(* LS Electric XG5000 project: 232통신_테스트 *)
(* PLC NewPLC *)
(* module base 0 slot 0: FEnet:XGL-EFMT(B) (Fast Ethernet 통신 모듈, 전기 Master) *)
(* module base 0 slot 1: Cnet:XGL-CH2A/B (Cnet 통신 모듈(RS-232C, RS-422/485)) *)
(* module base 0 slot 2: 입력 모듈:XGI-D22A/B (DC 24V 입력, 16점 (전류소스 싱크공용/ 전류소스 입력)) *)
(* module base 0 slot 3: 출력 모듈:XGQ-RY2A/B (릴레이 출력, 16점 (2A용, Varistor 없음/Varistor 부착)) *)

PROGRAM 메인 (* task: 스캔 프로그램 *)
VAR
    timer : TON;
    WATER_TIMER : TON;
    남은금액_1 : UINT;
    남은금액_2 : UINT;
    반환_타이머 : BOOL;
    사이다_TIMER : TON;
    식혜_TIMER : TON;
    알로에_TIMER : TON;
    자판기_거스름돈갯수_100원 AT %MW123 : UINT; (* 자판기_거스름돈갯수_100원 *)
    자판기_거스름돈갯수_500원 AT %MW122 : UINT; (* 자판기_거스름돈갯수_500원 *)
    자판기_거스름돈갯수_50원 AT %MW124 : UINT; (* 자판기_거스름돈갯수_50원 *)
    자판기_금액투입_1000원 AT %MW100.0 : BOOL; (* 자판기_금액투입_1000원 *)
    자판기_금액투입_100원 AT %MW100.2 : BOOL; (* 자판기_금액투입_100원 *)
    자판기_금액투입_500원 AT %MW100.1 : BOOL; (* 자판기_금액투입_500원 *)
    자판기_금액투입_50원 AT %MW100.3 : BOOL; (* 자판기_금액투입_50원 *)
    자판기_남은금액 AT %MW121 : UINT; (* 자판기_남은금액 *)
    자판기_물구매_700원 AT %MW100.5 : BOOL; (* 자판기_물구매_700원 *)
    자판기_반환버튼 AT %MW100.4 : BOOL; (* 자판기_반환버튼 *)
    자판기_사이다구매_1000원 AT %MW100.6 : BOOL; (* 자판기_사이다구매_1000원 *)
    자판기_식혜구매_1200원 AT %MW100.8 : BOOL; (* 자판기_식혜구매_1200원 *)
    자판기_알로에구매_1300원 AT %MW100.9 : BOOL; (* 자판기_알로에구매_1300원 *)
    자판기_음료출몰_물 AT %MW110.4 : BOOL; (* 자판기_음료출몰_물 *)
    자판기_음료출몰_사이다 AT %MW110.5 : BOOL; (* 자판기_음료출몰_사이다 *)
    자판기_음료출몰_식혜 AT %MW110.7 : BOOL; (* 자판기_음료출몰_식혜 *)
    자판기_음료출몰_알로에 AT %MW110.8 : BOOL; (* 자판기_음료출몰_알로에 *)
    자판기_음료출몰_콜라 AT %MW110.6 : BOOL; (* 자판기_음료출몰_콜라 *)
    자판기_콜라구매_1000원 AT %MW100.7 : BOOL; (* 자판기_콜라구매_1000원 *)
    자판기_투입금액 AT %MW120 : UINT; (* 자판기_투입금액 *)
    자판기램프_물 AT %MW110.0 : BOOL; (* 자판기램프_물 *)
    자판기램프_사이다_콜라 AT %MW110.1 : BOOL; (* 자판기램프_사이다_콜라 *)
    자판기램프_식혜 AT %MW110.2 : BOOL; (* 자판기램프_식혜 *)
    자판기램프_알로에 AT %MW110.3 : BOOL; (* 자판기램프_알로에 *)
    콜라_TIMER : TON;
END_VAR
VAR
    _e1 : R_TRIG;
    _e2 : R_TRIG;
    _e3 : R_TRIG;
    _e4 : R_TRIG;
    _e5 : R_TRIG;
    _e6 : R_TRIG;
    _t7 : BOOL;
    _e8 : R_TRIG;
    _t9 : BOOL;
    _t10 : BOOL;
    _e11 : R_TRIG;
    _t12 : BOOL;
    _e13 : R_TRIG;
    _e14 : F_TRIG;
    _e15 : R_TRIG;
    _t16 : BOOL;
    _e17 : R_TRIG;
    _t18 : BOOL;
    _e19 : R_TRIG;
    _t20 : BOOL;
    _e21 : R_TRIG;
    _t22 : BOOL;
    _e23 : R_TRIG;
    _t24 : BOOL;
END_VAR

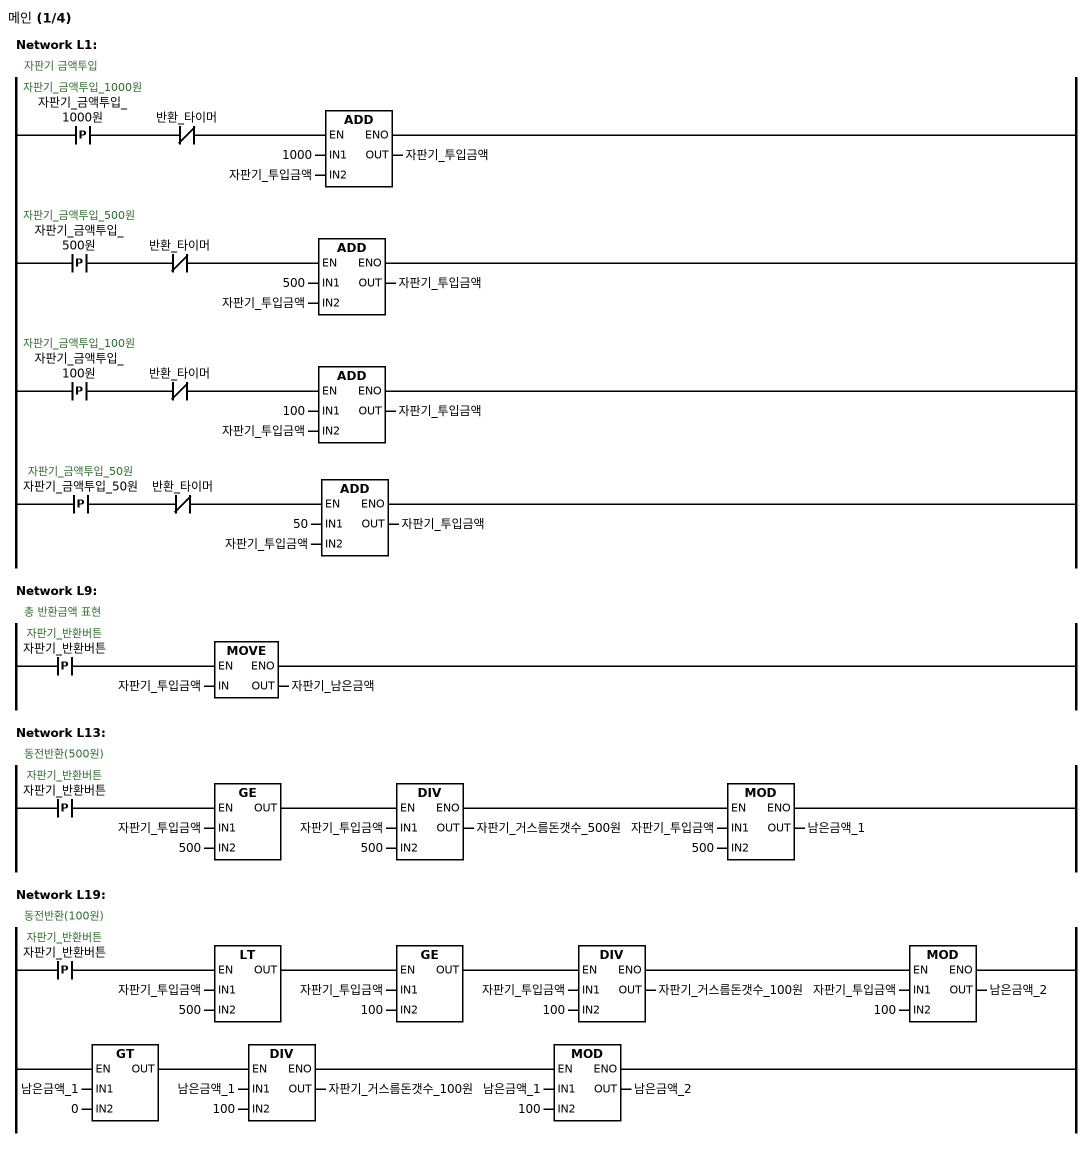
(* 자판기 금액투입 *)
(* Rung L1 *)
_e1(CLK := 자판기_금액투입_1000원);
IF _e1.Q AND NOT 반환_타이머 THEN 자판기_투입금액 := 1000 + 자판기_투입금액; END_IF;
_e2(CLK := 자판기_금액투입_500원);
IF _e2.Q AND NOT 반환_타이머 THEN 자판기_투입금액 := 500 + 자판기_투입금액; END_IF;
_e3(CLK := 자판기_금액투입_100원);
IF _e3.Q AND NOT 반환_타이머 THEN 자판기_투입금액 := 100 + 자판기_투입금액; END_IF;
_e4(CLK := 자판기_금액투입_50원);
IF _e4.Q AND NOT 반환_타이머 THEN 자판기_투입금액 := 50 + 자판기_투입금액; END_IF;
(* 총 반환금액 표현 *)
(* Rung L9 *)
_e5(CLK := 자판기_반환버튼);
IF _e5.Q THEN 자판기_남은금액 := 자판기_투입금액; END_IF;
(* 동전반환(500원) *)
(* Rung L13 *)
_e6(CLK := 자판기_반환버튼);
IF _e6.Q THEN _t7 := 자판기_투입금액 >= 500; END_IF;
IF _t7 THEN
    자판기_거스름돈갯수_500원 := 자판기_투입금액 / 500;
    남은금액_1 := 자판기_투입금액 MOD 500;
END_IF;
(* 동전반환(100원) *)
(* Rung L19 *)
_e8(CLK := 자판기_반환버튼);
IF _e8.Q THEN _t9 := 자판기_투입금액 < 500; END_IF;
IF _t9 THEN _t10 := 자판기_투입금액 >= 100; END_IF;
IF _t10 THEN
    자판기_거스름돈갯수_100원 := 자판기_투입금액 / 100;
    남은금액_2 := 자판기_투입금액 MOD 100;
END_IF;
IF 남은금액_1 > 0 THEN
    자판기_거스름돈갯수_100원 := 남은금액_1 / 100;
    남은금액_2 := 남은금액_1 MOD 100;
END_IF;

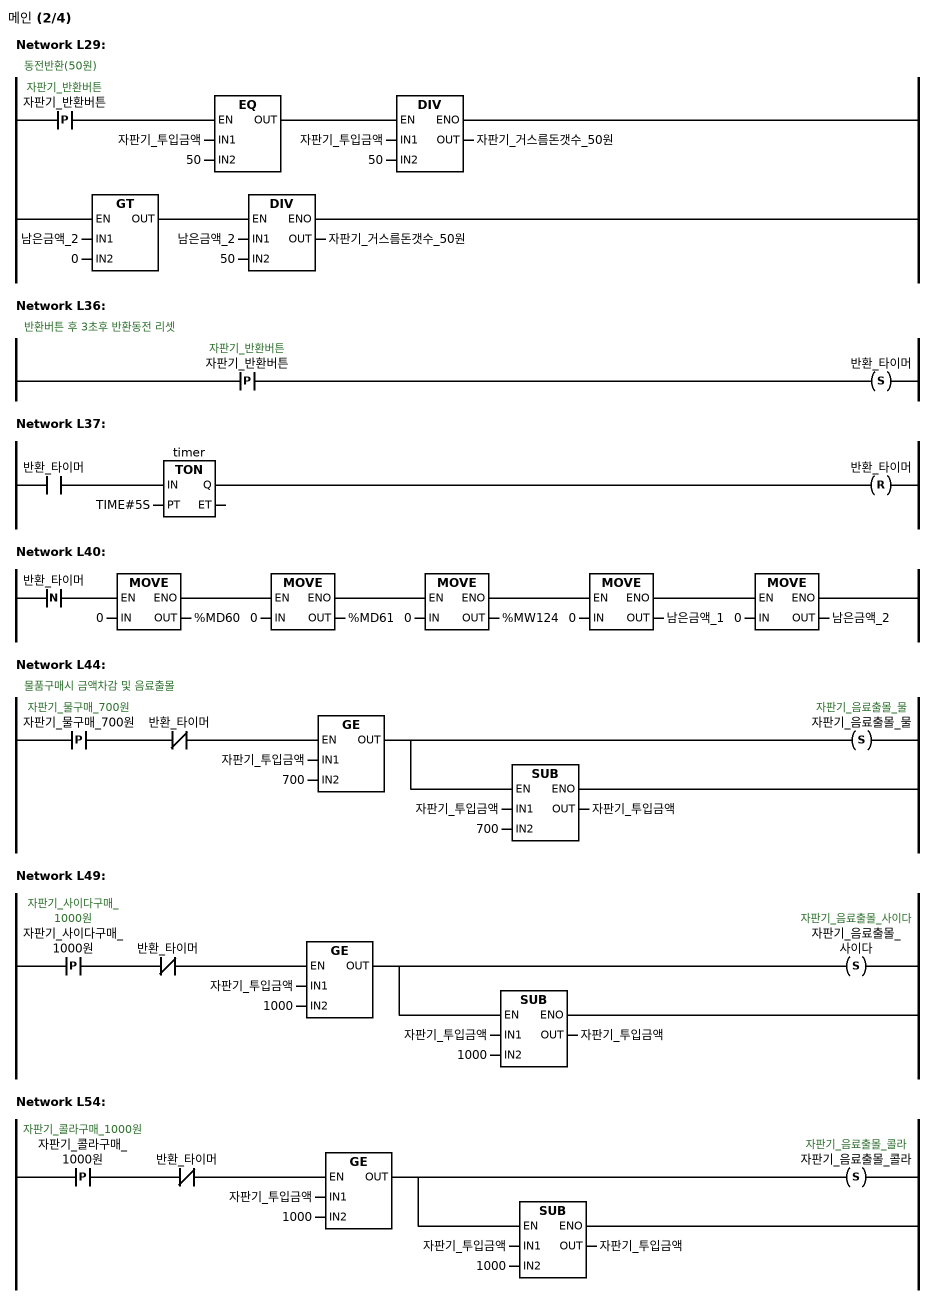
(* 동전반환(50원) *)
(* Rung L29 *)
_e11(CLK := 자판기_반환버튼);
IF _e11.Q THEN _t12 := 자판기_투입금액 = 50; END_IF;
IF _t12 THEN 자판기_거스름돈갯수_50원 := 자판기_투입금액 / 50; END_IF;
IF 남은금액_2 > 0 THEN 자판기_거스름돈갯수_50원 := 남은금액_2 / 50; END_IF;
(* 반환버튼 후 3초후 반환동전 리셋 *)
(* Rung L36 *)
_e13(CLK := 자판기_반환버튼);
IF _e13.Q THEN 반환_타이머 := TRUE; END_IF;
(* Rung L37 *)
timer(IN := 반환_타이머, PT := TIME#5S);
IF timer.Q THEN 반환_타이머 := FALSE; END_IF;
(* Rung L40 *)
_e14(CLK := 반환_타이머);
IF _e14.Q THEN
    %MD60 := 0;
    %MD61 := 0;
    %MW124 := 0;
    남은금액_1 := 0;
    남은금액_2 := 0;
END_IF;
(* 물품구매시 금액차감 및 음료출몰 *)
(* Rung L44 *)
_e15(CLK := 자판기_물구매_700원);
IF _e15.Q AND NOT 반환_타이머 THEN _t16 := 자판기_투입금액 >= 700; END_IF;
IF _t16 THEN
    자판기_음료출몰_물 := TRUE;
    자판기_투입금액 := 자판기_투입금액 - 700;
END_IF;
(* Rung L49 *)
_e17(CLK := 자판기_사이다구매_1000원);
IF _e17.Q AND NOT 반환_타이머 THEN _t18 := 자판기_투입금액 >= 1000; END_IF;
IF _t18 THEN
    자판기_음료출몰_사이다 := TRUE;
    자판기_투입금액 := 자판기_투입금액 - 1000;
END_IF;
(* Rung L54 *)
_e19(CLK := 자판기_콜라구매_1000원);
IF _e19.Q AND NOT 반환_타이머 THEN _t20 := 자판기_투입금액 >= 1000; END_IF;
IF _t20 THEN
    자판기_음료출몰_콜라 := TRUE;
    자판기_투입금액 := 자판기_투입금액 - 1000;
END_IF;

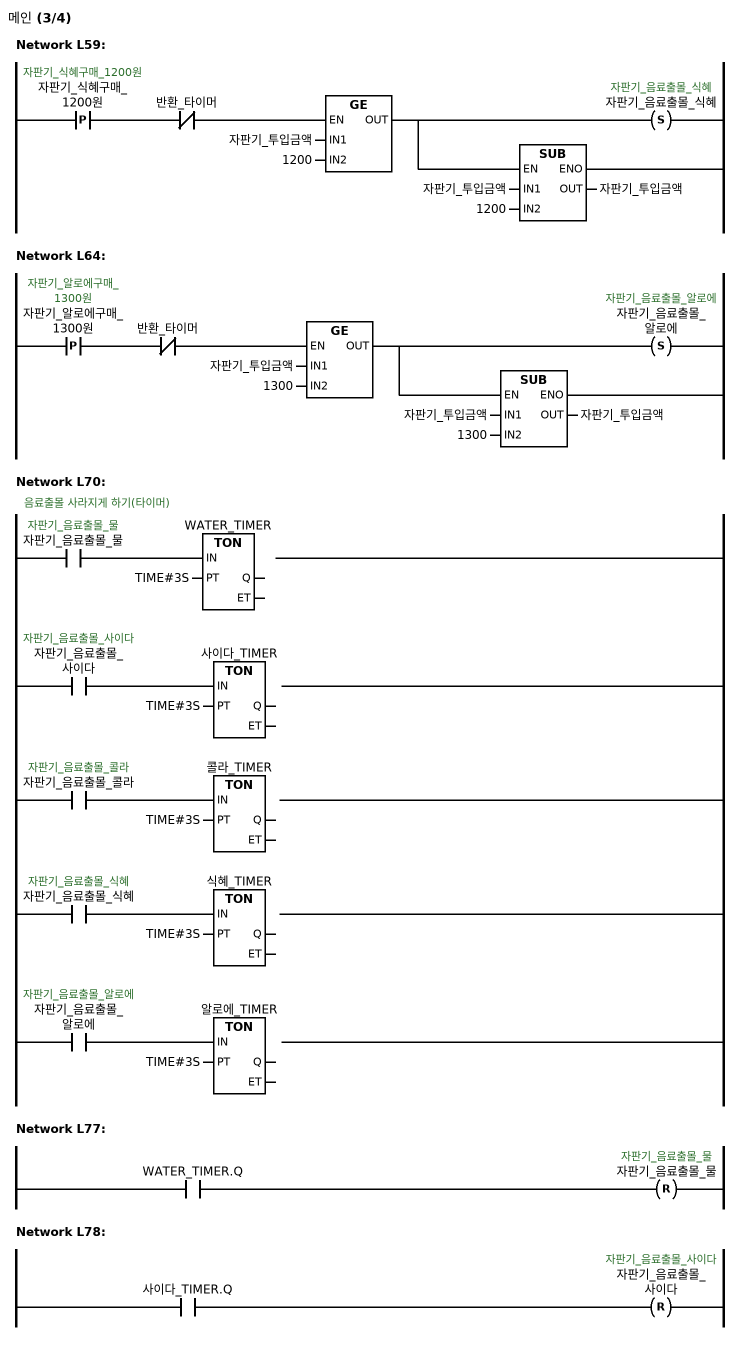
(* Rung L59 *)
_e21(CLK := 자판기_식혜구매_1200원);
IF _e21.Q AND NOT 반환_타이머 THEN _t22 := 자판기_투입금액 >= 1200; END_IF;
IF _t22 THEN
    자판기_음료출몰_식혜 := TRUE;
    자판기_투입금액 := 자판기_투입금액 - 1200;
END_IF;
(* Rung L64 *)
_e23(CLK := 자판기_알로에구매_1300원);
IF _e23.Q AND NOT 반환_타이머 THEN _t24 := 자판기_투입금액 >= 1300; END_IF;
IF _t24 THEN
    자판기_음료출몰_알로에 := TRUE;
    자판기_투입금액 := 자판기_투입금액 - 1300;
END_IF;
(* 음료출몰 사라지게 하기(타이머) *)
(* Rung L70 *)
WATER_TIMER(IN := 자판기_음료출몰_물, PT := TIME#3S);
사이다_TIMER(IN := 자판기_음료출몰_사이다, PT := TIME#3S);
콜라_TIMER(IN := 자판기_음료출몰_콜라, PT := TIME#3S);
식혜_TIMER(IN := 자판기_음료출몰_식혜, PT := TIME#3S);
알로에_TIMER(IN := 자판기_음료출몰_알로에, PT := TIME#3S);
(* Rung L77 *)
IF WATER_TIMER.Q THEN 자판기_음료출몰_물 := FALSE; END_IF;
(* Rung L78 *)
IF 사이다_TIMER.Q THEN 자판기_음료출몰_사이다 := FALSE; END_IF;

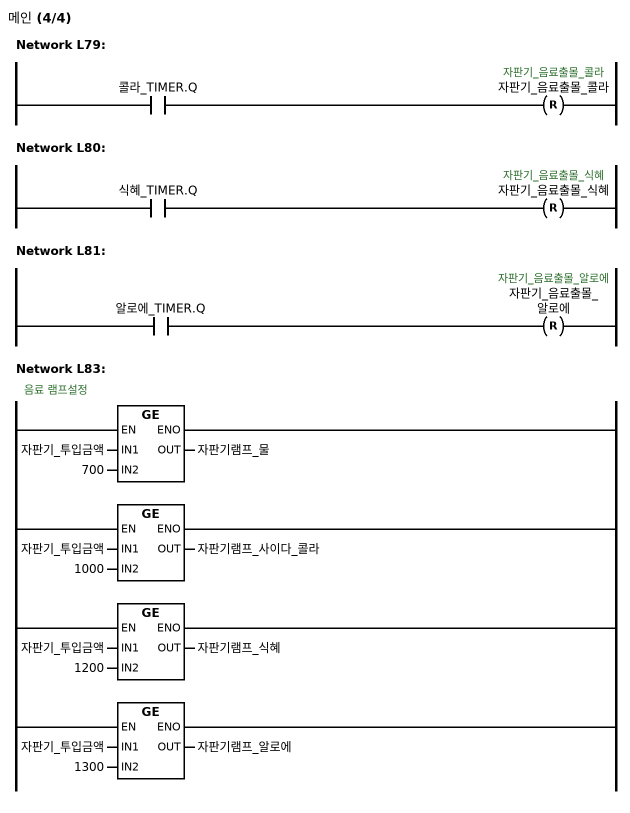
(* Rung L79 *)
IF 콜라_TIMER.Q THEN 자판기_음료출몰_콜라 := FALSE; END_IF;
(* Rung L80 *)
IF 식혜_TIMER.Q THEN 자판기_음료출몰_식혜 := FALSE; END_IF;
(* Rung L81 *)
IF 알로에_TIMER.Q THEN 자판기_음료출몰_알로에 := FALSE; END_IF;
(* 음료 램프설정 *)
(* Rung L83 *)
자판기램프_물 := 자판기_투입금액 >= 700;
자판기램프_사이다_콜라 := 자판기_투입금액 >= 1000;
자판기램프_식혜 := 자판기_투입금액 >= 1200;
자판기램프_알로에 := 자판기_투입금액 >= 1300;
END_PROGRAM